{attribute 'qualified_only'}
{attribute 'strict'}
TYPE E_CNC_Robot_Path :
(
	NoPath,
	Lift1A_to_CNC1,
	Lift1B_to_CNC1,
	CNC1_to_Lift1A,
	CNC1_to_Lift1B,
	Lift2A_to_CNC2,
	Lift2B_to_CNC2,
	CNC2_to_Lift2A,
	CNC2_to_Lift2B,
	Lift3A_to_CNC3,
	Lift3B_to_CNC3,
	CNC3_to_Lift3A,
	CNC3_to_Lift3B
);
END_TYPE

(* stored: Version 1.1.0.1, ProductVersion 3.1.4024.12
   EnumerationTextList E_CNC_Robot_Path: Id {2ebe0acd-70e6-4b67-98e1-dd0f2591f869} *)
